// Bunker HMI interface - ONE struct per tile.
//
// Extends ST_ComponentBase_HMI, so Config, Command and Status arrive inherited
// and the added members cannot reuse those three names.
TYPE ST_AbstractBunker_HMI EXTENDS ST_ComponentBase_HMI :
STRUCT
	DeviceCommand	: ST_AbstractBunker_Command;
	Device			: ST_AbstractBunker_Status;
END_STRUCT
END_TYPE

(* stored: Version 1.1.0.1, ProductVersion 3.1.4026.19
   DUT ST_AbstractBunker_HMI: Id {d8898eee-1ff7-487f-b9a3-8d65837f3b26} *)
